// TIA Portal V19 export
TYPE "lexchangetray_typeUnEmnTranserfCondition"
// Type: Bool
// stored: Access Published
   STRUCT
      axisPosMoveCondition : Bool;
   END_STRUCT;
END_TYPE
